FUNCTION_BLOCK FB_VacuumValve
VAR_INPUT
	ValveTime : TIME := T#500MS;
	ETime : TIME := T#0MS;
	CalcTime : TIME := T#500MS;
END_VAR
VAR_OUTPUT
END_VAR
VAR_IN_OUT
	stAVol : ST_Volume;
	stBVol : ST_Volume;
	stValve : ST_VacuumValve;
END_VAR
VAR
	ClsTOF:TOF;
	OpnTON:TON;
	ClsInverter : BOOL;
	r_t : R_TRIG;
	f_t : F_TRIG;
	State : INT;
	//calculates prevous times to send correct PT
	CalcOpenTime : TIME := T#0MS;
END_VAR

(* 
Vacuum Valve Simulation

A valve has two ports, A and B.
And two states, open or closed. (transition = open)
Valve open:
Average of A and B is written to both sides.

Limit switches
Solenoid goes high:
1. Normal switch goes low
2. Timer for motion elapses
3. Actuated switch goes high

2017-2-17 A. Pai
*)

(* Pressure transfer *)
IF NOT stValve.q_xClsLS THEN
	stBVol.rPressure := (stAVol.rPressure*stAVol.rVolume + stBVol.rPressure*stBVol.rVolume)/(stAVol.rVolume+stBVol.rVolume);
	stAVol.rPressure := stBVol.rPressure;
END_IF

(* Valve motion *)
OpnTON.IN := stValve.i_xSol;
r_t(CLK := stValve.i_xSol); 

ClsTOF.IN := stValve.i_xSol;
f_t(CLK := stValve.i_xSol);

//If there is a rising edge then change OpnTON.PT
IF(r_t.Q)THEN
	IF State = 0 THEN
	CalcOpenTime := ValveTime;
	END_IF
	// if previous state = 2
	IF State = 2 THEN
		CalcOpenTime := CalcOpenTime + ClsTOF.ET;
	END_IF
	OpnTON.PT := CalcOpenTime;
	//set state = 1 for rising edge case
	State := 1;
END_IF

//If there is a falling edge then change ClsTOF.PT
IF(f_t.Q) THEN
	IF State = 0 THEN
	CalcOpenTime := T#0MS;
	END_IF
	// if previous state = 1
	IF State = 1 THEN
		CalcOpenTime := OpnTON.ET - CalcOpenTime ;
		//ClsTOF.PT := ValveTime - CalcOpenTime;
	END_IF
	ClsTOF.PT := ValveTime - CalcOpenTime;
	//set state = 2 for falling edge case
	State := 2;
END_IF

//run both TON and TOF timers 
OpnTON(Q=>stValve.q_xOpnLS);
ClsTOF(Q=>ClsInverter);

//Invert signal to correct value
stValve.q_xClsLS := NOT ClsInverter;

//If open and close values stablized then set ETime to 0ms
IF(stValve.q_xOpnLS XOR stValve.q_xClsLS) THEN
	// reset CalcOpenTime
	//CalcOpenTime := T#0MS;
	// stable state
	State := 0;
END_IF

END_FUNCTION_BLOCK

(* stored: Version 1.1.0.1, ProductVersion 3.1.4020.12
   POU FB_VacuumValve: Id {2e26d57b-cfa8-4953-9619-5535d3a3ce01}, SpecialFunc None *)
